TYPE ST_Xbox_2D_Joystick_NC_Options :
STRUCT
	// Inverts the direction of the X axis
	bInverted_X : BOOL := FALSE;
	// Inverts the direction of the Y axis
	bInverted_Y : BOOL := FALSE;
	// Maximum Feedrate X Axis
	fMaxOverride_X : LREAL := 100.0;
	// Maximum Feedrate Y Axis
	fMaxOverride_Y : LREAL := 100.0;
	// Struct of parameters for MC_Halt command
	stXbox_NC_Halt_Dynamics : ST_Xbox_NC_Halt_Dynamics;
END_STRUCT
END_TYPE

(* stored: Version 1.1.0.1, ProductVersion 3.1.4024.11
   DUT ST_Xbox_2D_Joystick_NC_Options: Id {33988ec7-80f6-4620-9e26-ff99c54086ea} *)
